TYPE "MEStoPLC_MainCheckOut"
VERSION : 0.1
   STRUCT
      "M-DataSaveDone" : Bool;
      "M-DataSaveOK" : Bool;
      "M-DataSaveNG" : Bool;
      "M-DataSaveErrCode" : Int;
      "M-DataSaveErrMsg" : String[98];
      Reserve : Array[1..2096] of Byte;
   END_STRUCT;

END_TYPE

